// TIA Portal V17 export
// export: Created 2024-09-02T12:50:30.4240342Z, ExportSetting WithDefaults, DisplayName Totally Integrated Automation Portal, DisplayVersion V17, DisplayName TIA Portal Openness, DisplayVersion V17, DisplayName TIA Portal Version Control Interface, DisplayVersion V17, DisplayName STEP 7 Professional, DisplayVersion V17, DisplayName STEP 7 Safety, DisplayVersion V17, DisplayName WinCC Professional, DisplayVersion V17
TYPE "type_Cognex_VS"
// stored: IsFailsafeCompliant false
   STRUCT
      HMI : Struct   // HMI-Button
         FrgFkt : Struct   // Freigabe / Approve
            Gestaltung : Int;   // Button Anzeige Gestaltung / Button Display Design
            aktiv : Bool;   // Button aktiv (gedrückt) / Button active (pressed)
         END_STRUCT;
         Reset : Struct   // Button "Reset"
            Gestaltung : Int;   // Button Anzeige Gestaltung / Button Display Design
            aktiv : Bool;   // Button aktiv (gedrückt) / Button active (pressed)
         END_STRUCT;
         Read : Struct   // Button "Read"
            Gestaltung : Int;   // Button Anzeige Gestaltung / Button Display Design
            aktiv : Bool;   // Button aktiv (gedrückt) / Button active (pressed)
         END_STRUCT;
         SetPrg : Struct   // Button "Set Programm"
            Gestaltung : Int;   // Button Anzeige Gestaltung / Button Display Design
            aktiv : Bool;   // Button aktiv (gedrückt) / Button active (pressed)
         END_STRUCT;
         Write : Struct   // Button "Write"
            Gestaltung : Int;   // Button Anzeige Gestaltung / Button Display Design
            aktiv : Bool;   // Button aktiv (gedrückt) / Button active (pressed)
         END_STRUCT;
         Lighting : Struct   // Button "Lighting"
            Gestaltung : Int;   // Button Anzeige Gestaltung / Button Display Design
            aktiv : Bool;   // Button aktiv (gedrückt) / Button active (pressed)
         END_STRUCT;
         ResetStatistik : Struct   // Button "Statistik Reset"
            Gestaltung : Int;   // Button Anzeige Gestaltung / Button Display Design
            aktiv : Bool;   // Button aktiv (gedrückt) / Button active (pressed)
         END_STRUCT;
         Res_07 : Struct   // Button " "
            Gestaltung : Int;   // Button Anzeige Gestaltung / Button Display Design
            aktiv : Bool;   // Button aktiv (gedrückt) / Button active (pressed)
         END_STRUCT;
         Res_08 : Struct   // Button " "
            Gestaltung : Int;   // Button Anzeige Gestaltung / Button Display Design
            aktiv : Bool;   // Button aktiv (gedrückt) / Button active (pressed)
         END_STRUCT;
         ProgNbr { S7_SetPoint := 'True'} : Int := 1;   // Program number for reset operation (default "1")
      END_STRUCT;
      Anzeige : Struct   // Anzeige / Display
         StatusBool { ExternalWritable := 'False'} : DWord;   // Status
         StatusInt { ExternalWritable := 'False'} : Array[0..5] of Int;   // Status ID / status ID
         Ergebnis { ExternalWritable := 'False'} : Array[0..7] of LInt;   // Statistik / Statistics
      END_STRUCT;
      Start { ExternalWritable := 'False'} : Bool;   // Start
      Reset { ExternalWritable := 'False'} : Bool;   // Reset
      Licht { ExternalWritable := 'False'} : Bool;   // Licht ein / Light on
      Done { ExternalWritable := 'False'} : Bool;   // Kamera Done / Camera Done
      DoneFl { ExternalWritable := 'False'} : Bool;   // Kamera Done Flanke / Camera Done flank
      Result_IO { ExternalWritable := 'False'} : Bool;   // Kamera Result IO / Camera Result IO
      Result_IO_1 { ExternalWritable := 'False'} : Bool;   // Kamera Result Code 1 IO / Camera Result Code 1 IO
      Result_IO_2 { ExternalWritable := 'False'} : Bool;   // Kamera Result Code 2 IO / Camera Result Code 2 IO
      Error { ExternalWritable := 'False'} : Byte;   // Result error in written result (match error, read error) / Result error in written result (match error, read error)
      ProgNr { ExternalWritable := 'False'} : Int;   // Programmnummer / program number
      ResultQ { ExternalWritable := 'False'} : Char;   // Code quality / Code quality
      ResultLn { ExternalWritable := 'False'} : Int;   // Anzahl Daten / Number of data:
      ResultStr { ExternalWritable := 'False'} : String;   // Daten in String / Data in string
      InDaten { ExternalWritable := 'False'} : Struct   // Eingabedaten / input data
         StationsNr { ExternalWritable := 'False'} : Array[1..6] of Char;   // Adr.16
         KameraNr { ExternalWritable := 'False'} : Array[1..2] of Char;   // Adr.22
         PID { ExternalWritable := 'False'} : Array[1..30] of Char;   // Adr.24
         MotNr { ExternalWritable := 'False'} : Array[1..12] of Char;   // Adr.54
         ProgrammNr { ExternalWritable := 'False'} : Array[1..2] of Char;   // Adr.66
         ErweiterteDaten { ExternalWritable := 'False'} : Array[1..30] of Char;   // Adr.68
         Res { ExternalWritable := 'False'} : Array[98..127] of Char;
      END_STRUCT;
      Scanndaten { ExternalWritable := 'False'} : Struct   // Scanndaten / scanning data
         Code_1 { ExternalWritable := 'False'} : Array[1..100] of Char;   // Eingabedaten / input data
         Code_2 { ExternalWritable := 'False'} : Array[1..100] of Char;   // Eingabedaten / input data
      END_STRUCT;
      DatenChar { ExternalWritable := 'False'} : Struct   // Ergebnissdaten in Char / Result data in Char
         ED { ExternalWritable := 'False'} : Array[1..58] of Char;
      END_STRUCT;
      DatenDez { ExternalWritable := 'False'} : Struct   // Ergebnissdaten in Dezimal / Result data in decimal
         ED { ExternalWritable := 'False'} : Array[1..58] of Byte;
      END_STRUCT;
   END_STRUCT;
END_TYPE
